# EPICS autosave request: tests/testfiles/cfg/SF_OpticsMBND_PV.req
$(SYS):ONOFF
$(SYS):K0L-SET
